(* PLC project Unnamed, Unknown Unnamed 1 *)
(* stored: creationDateTime 2026-03-24T22:18:36, modificationDateTime 2026-05-19T17:14:10 *)

PROGRAM Exercise5
  VAR
    Left_Hand AT %QX0.0 : BOOL;
    Right_Hand AT %QX0.1 : BOOL;
    Guard_Front AT %QX0.2 : BOOL;
    Guard_Left AT %QX0.3 : BOOL;
    Guard_Right AT %QX0.4 : BOOL;
    E_Stop AT %QX0.5 : BOOL;
    Mode_Switch AT %QX1.0 : BOOL;
    Key_Switch AT %QX1.1 : BOOL;
    Stroke_Sensor AT %QX1.2 : BOOL;
    Pressure_Pump AT %QX1.3 : BOOL;
    Press_Ram_Full AT %QX1.4 : BOOL;
    Press_Ram_Slow AT %QX1.5 : BOOL;
    Safety_OK AT %QX1.6 : BOOL;
    Fault_Light AT %QX1.7 : BOOL;
    Pump_Run_Light AT %QX2.0 : BOOL;
    Jam_Fault_Light AT %QX2.1 : BOOL;
    Stabilization_Done AT %MX0.0 : BOOL;
    Prev_Mode AT %MX0.1 : BOOL;
    Mode_Changed AT %MX0.2 : BOOL;
    Both_Hands AT %MX0.3 : BOOL;
  END_VAR
  VAR
    TON0 : TON;
    TON1 : TON;
  END_VAR

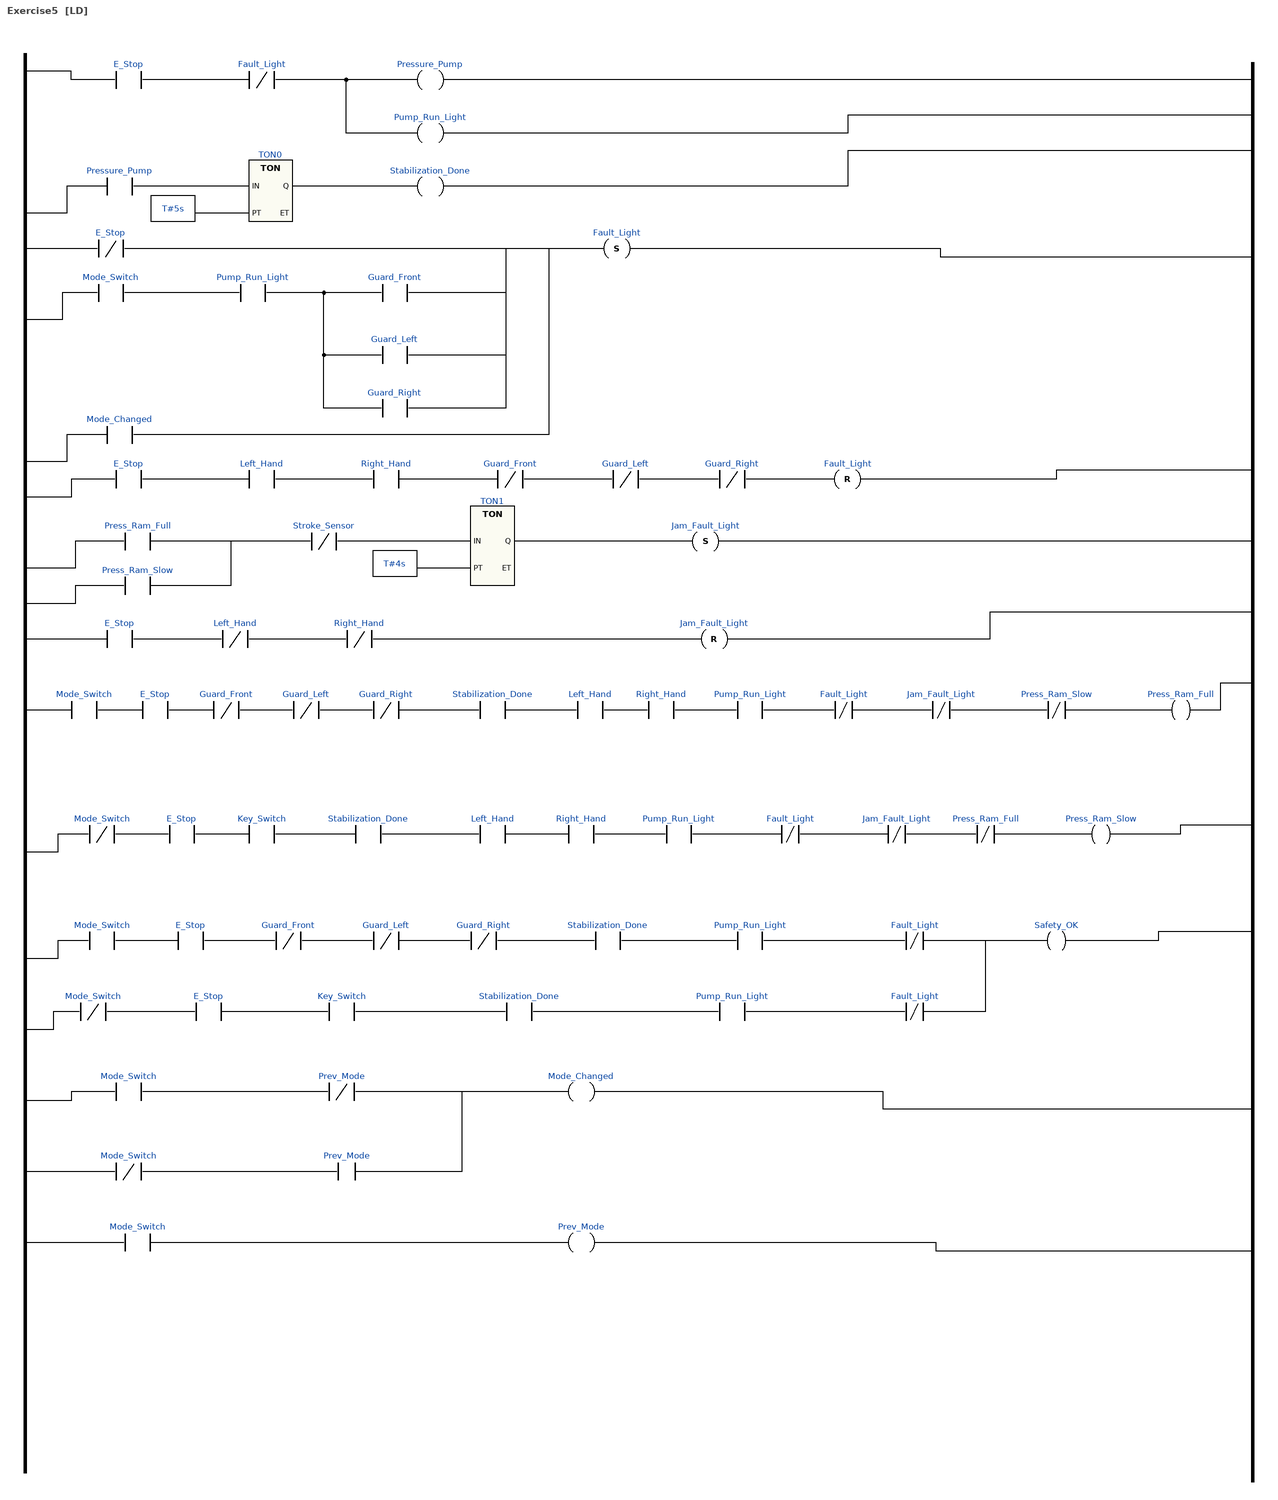
(* LD diagram, written out as Structured Text *)
Pressure_Pump := E_Stop AND NOT Fault_Light;
Pump_Run_Light := E_Stop AND NOT Fault_Light;
TON0(IN := Pressure_Pump, PT := T#5s);
Stabilization_Done := TON0.Q;
IF E_Stop AND Left_Hand AND Right_Hand AND NOT Guard_Front AND NOT Guard_Left AND NOT Guard_Right THEN Fault_Light := FALSE; END_IF;
IF NOT E_Stop OR Mode_Switch AND Pump_Run_Light AND Guard_Front OR Mode_Switch AND Pump_Run_Light AND Guard_Left OR Mode_Switch AND Pump_Run_Light AND Guard_Right OR Mode_Changed THEN Fault_Light := TRUE; END_IF;
TON1(IN := (Press_Ram_Full OR Press_Ram_Slow) AND NOT Stroke_Sensor, PT := T#4s);
IF TON1.Q THEN Jam_Fault_Light := TRUE; END_IF;
IF E_Stop AND NOT Left_Hand AND NOT Right_Hand THEN Jam_Fault_Light := FALSE; END_IF;
Press_Ram_Full := Mode_Switch AND E_Stop AND NOT Guard_Front AND NOT Guard_Left AND NOT Guard_Right AND Stabilization_Done AND Left_Hand AND Right_Hand AND Pump_Run_Light AND NOT Fault_Light AND NOT Jam_Fault_Light AND NOT Press_Ram_Slow;
Press_Ram_Slow := NOT Mode_Switch AND E_Stop AND Key_Switch AND Stabilization_Done AND Left_Hand AND Right_Hand AND Pump_Run_Light AND NOT Fault_Light AND NOT Jam_Fault_Light AND NOT Press_Ram_Full;
Safety_OK := Mode_Switch AND E_Stop AND NOT Guard_Front AND NOT Guard_Left AND NOT Guard_Right AND Stabilization_Done AND Pump_Run_Light AND NOT Fault_Light OR NOT Mode_Switch AND E_Stop AND Key_Switch AND Stabilization_Done AND Pump_Run_Light AND NOT Fault_Light;
Mode_Changed := Mode_Switch AND NOT Prev_Mode OR NOT Mode_Switch AND Prev_Mode;
Prev_Mode := Mode_Switch;
END_PROGRAM

CONFIGURATION Config0
  RESOURCE Res0 ON PLC
    TASK task0(INTERVAL := T#20ms, PRIORITY := 0);
    PROGRAM instance0 WITH task0 : Exercise5;
  END_RESOURCE
END_CONFIGURATION
